TYPE ST_InputStationHSAdditionalDataOP11600 :
STRUCT
	{attribute 'OPC.UA.DA.Description' := 'Initial Temperature'}
	TempInitial					: REAL := 20.0;

END_STRUCT
END_TYPE

(* stored: Version 1.1.0.1, ProductVersion 3.1.4024.5
   DUT ST_InputStationHSAdditionalDataOP11600: Id {8a95d514-54fb-4306-bc25-2f4f6b00cdbe} *)
